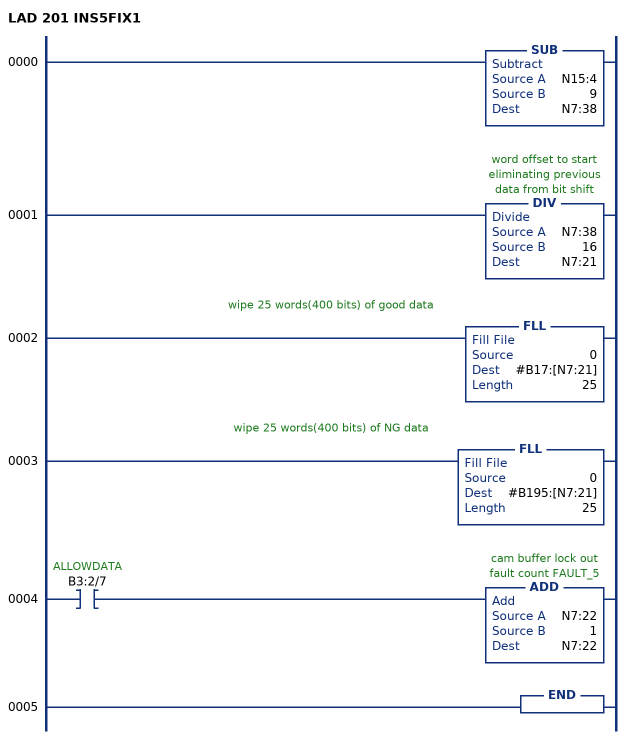
% Rung: 0 %
SOR SUB N15:4 9 N7:38 EOR
%   N15:4  INS_5_TRIG_LOC %
% Rung: 1 %
SOR DIV N7:38 16 N7:21 EOR
%   N7:21  "word offset to start eliminating previous data from bit shift" %
% Rung: 2 %
% wipe 25 words(400 bits) of good data %
SOR FLL 0 #B17:[N7:21] 25 EOR
%   N7:21  "word offset to start eliminating previous data from bit shift" %
% Rung: 3 %
% wipe 25 words(400 bits) of NG data %
SOR FLL 0 #B195:[N7:21] 25 EOR
%   N7:21  "word offset to start eliminating previous data from bit shift" %
% Rung: 4 %
SOR XIC B3:2/7 ADD N7:22 1 N7:22 EOR
%   B3:2/7  ALLOWDATA %
%   N7:22  FAULT_5  "cam buffer lock out fault count" %
% Rung: 5 %
SOR END EOR

LADDER 202 "INS5FIX2"
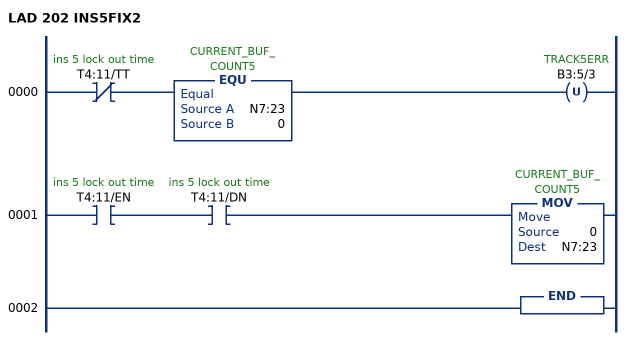
% Rung: 0 %
SOR XIO T4:11/TT EQU N7:23 0 OTU B3:5/3 EOR
%   T4:11  "ins 5 lock out time" %
%   N7:23  CURRENT_BUF_COUNT5 %
%   B3:5/3  TRACK5ERR %
% Rung: 1 %
SOR XIC T4:11/EN XIC T4:11/DN MOV 0 N7:23 EOR
%   T4:11  "ins 5 lock out time" %
%   N7:23  CURRENT_BUF_COUNT5 %
% Rung: 2 %
SOR END EOR

LADDER 203 "HS TRIG5"
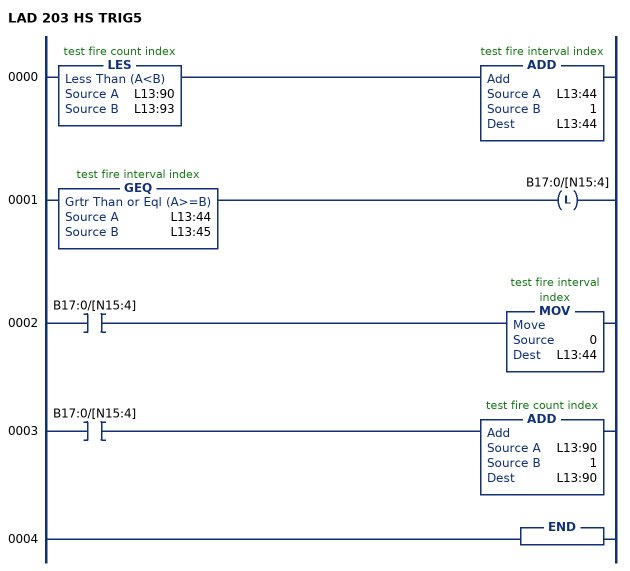
% Rung: 0 %
SOR LES L13:90 L13:93 ADD L13:44 1 L13:44 EOR
%   L13:90  "test fire count index" %
%   L13:93  "test fire count" %
%   L13:44  "test fire interval index" %
% Rung: 1 %
SOR GEQ L13:44 L13:45 OTL B17:0/[N15:4] EOR
%   L13:44  "test fire interval index" %
%   L13:45  "test fire interval" %
%   N15:4  INS_5_TRIG_LOC %
% Rung: 2 %
SOR XIC B17:0/[N15:4] MOV 0 L13:44 EOR
%   N15:4  INS_5_TRIG_LOC %
%   L13:44  "test fire interval index" %
% Rung: 3 %
SOR XIC B17:0/[N15:4] ADD L13:90 1 L13:90 EOR
%   N15:4  INS_5_TRIG_LOC %
%   L13:90  "test fire count index" %
% Rung: 4 %
SOR END EOR

LADDER 212 "INS6"
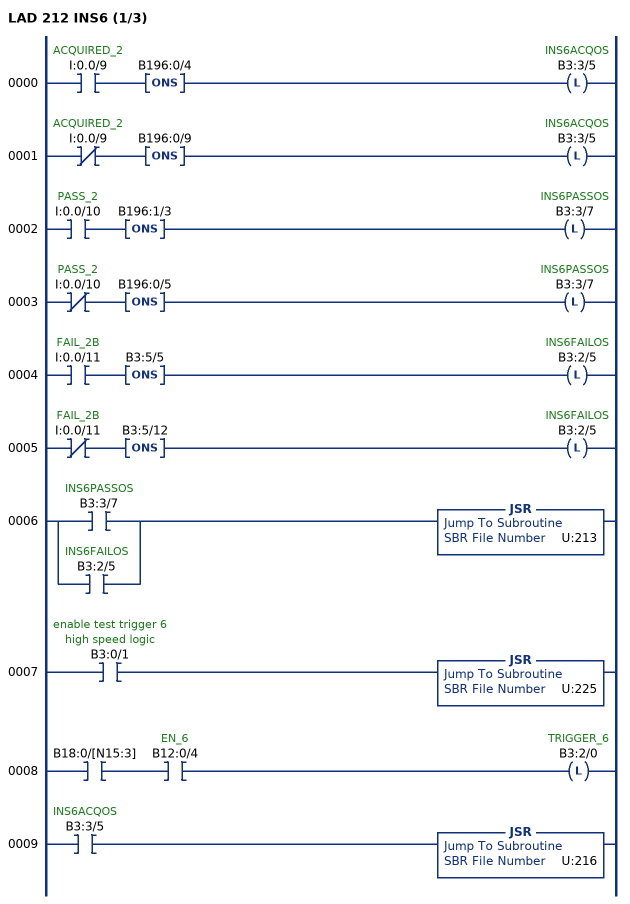
% Rung: 0 %
SOR XIC I:0.0/9 ONS B196:0/4 OTL B3:3/5 EOR
%   I:0.0/9  ACQUIRED_2 %
%   B3:3/5  INS6ACQOS %
% Rung: 1 %
SOR XIO I:0.0/9 ONS B196:0/9 OTL B3:3/5 EOR
%   I:0.0/9  ACQUIRED_2 %
%   B3:3/5  INS6ACQOS %
% Rung: 2 %
SOR XIC I:0.0/10 ONS B196:1/3 OTL B3:3/7 EOR
%   I:0.0/10  PASS_2 %
%   B3:3/7  INS6PASSOS %
% Rung: 3 %
SOR XIO I:0.0/10 ONS B196:0/5 OTL B3:3/7 EOR
%   I:0.0/10  PASS_2 %
%   B3:3/7  INS6PASSOS %
% Rung: 4 %
SOR XIC I:0.0/11 ONS B3:5/5 OTL B3:2/5 EOR
%   I:0.0/11  FAIL_2B %
%   B3:2/5  INS6FAILOS %
% Rung: 5 %
SOR XIO I:0.0/11 ONS B3:5/12 OTL B3:2/5 EOR
%   I:0.0/11  FAIL_2B %
%   B3:2/5  INS6FAILOS %
% Rung: 6 %
SOR BST XIC B3:3/7 NXB XIC B3:2/5 BND JSR U:213 EOR
%   B3:3/7  INS6PASSOS %
%   B3:2/5  INS6FAILOS %
% Rung: 7 %
SOR XIC B3:0/1 JSR U:225 EOR
%   B3:0/1  "enable test trigger 6 high speed logic" %
% Rung: 8 %
SOR XIC B18:0/[N15:3] XIC B12:0/4 OTL B3:2/0 EOR
%   N15:3  INS_6_TRIG_LOC %
%   B12:0/4  EN_6 %
%   B3:2/0  TRIGGER_6 %
% Rung: 9 %
SOR XIC B3:3/5 JSR U:216 EOR
%   B3:3/5  INS6ACQOS %

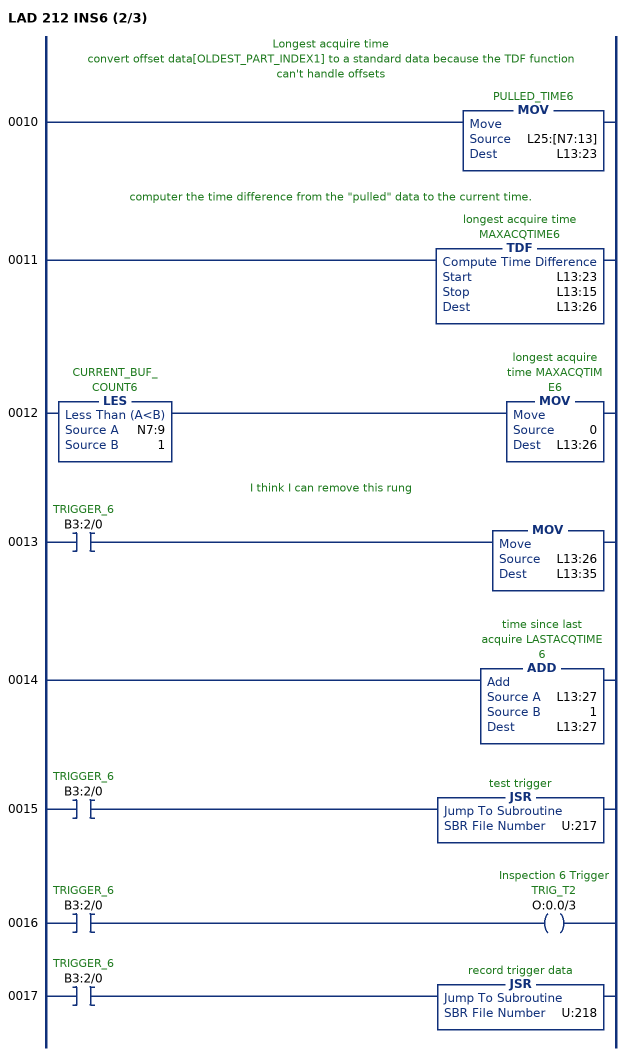
% Rung: 10 %
% Longest acquire time
% convert offset data[OLDEST_PART_INDEX1] to a standard data because the TDF function can't handle offsets %
SOR MOV L25:[N7:13] L13:23 EOR
%   N7:13  OLDEST_PART_INDEX6 %
%   L13:23  PULLED_TIME6 %
% Rung: 11 %
% computer the time difference from the "pulled" data to the current time. %
SOR TDF L13:23 L13:15 L13:26 EOR
%   L13:23  PULLED_TIME6 %
%   L13:15  TOP_TIME %
%   L13:26  MAXACQTIME6  "longest acquire time" %
% Rung: 12 %
SOR LES N7:9 1 MOV 0 L13:26 EOR
%   N7:9  CURRENT_BUF_COUNT6 %
%   L13:26  MAXACQTIME6  "longest acquire time" %
% Rung: 13 %
% I think I can remove this rung %
SOR XIC B3:2/0 MOV L13:26 L13:35 EOR
%   B3:2/0  TRIGGER_6 %
%   L13:26  MAXACQTIME6  "longest acquire time" %
% Rung: 14 %
SOR ADD L13:27 1 L13:27 EOR
%   L13:27  LASTACQTIME6  "time since last acquire" %
% Rung: 15 %
SOR XIC B3:2/0 JSR U:217 EOR
%   B3:2/0  TRIGGER_6 %
%   U:217  "test trigger" %
% Rung: 16 %
SOR XIC B3:2/0 OTE O:0.0/3 EOR
%   B3:2/0  TRIGGER_6 %
%   O:0.0/3  TRIG_T2  "Inspection 6 Trigger" %
% Rung: 17 %
SOR XIC B3:2/0 JSR U:218 EOR
%   B3:2/0  TRIGGER_6 %
%   U:218  "record trigger data" %

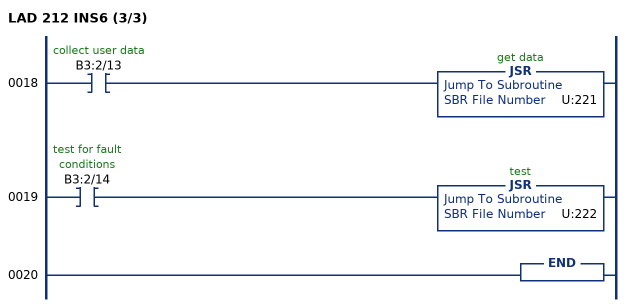
% Rung: 18 %
SOR XIC B3:2/13 JSR U:221 EOR
%   B3:2/13  "collect user data" %
%   U:221  "get data" %
% Rung: 19 %
SOR XIC B3:2/14 JSR U:222 EOR
%   B3:2/14  "test for fault conditions" %
%   U:222  "test" %
% Rung: 20 %
SOR END EOR

LADDER 213 "INS6RESULT"
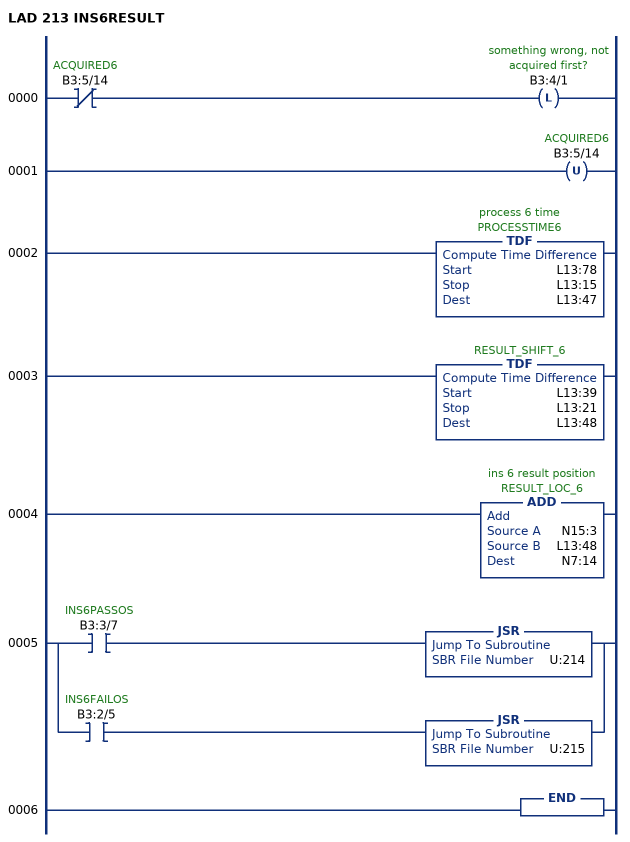
% Rung: 0 %
SOR XIO B3:5/14 OTL B3:4/1 EOR
%   B3:5/14  ACQUIRED6 %
%   B3:4/1  "something wrong, not acquired first?" %
% Rung: 1 %
SOR OTU B3:5/14 EOR
%   B3:5/14  ACQUIRED6 %
% Rung: 2 %
SOR TDF L13:78 L13:15 L13:47 EOR
%   L13:78  TIMEOFACQ6  "the time of the last acquire" %
%   L13:15  TOP_TIME %
%   L13:47  PROCESSTIME6  "process 6 time" %
% Rung: 3 %
SOR TDF L13:39 L13:21 L13:48 EOR
%   L13:39  PROCESS_START_POS_6 %
%   L13:21  TOP_POSITION %
%   L13:48  RESULT_SHIFT_6 %
% Rung: 4 %
SOR ADD N15:3 L13:48 N7:14 EOR
%   N15:3  INS_6_TRIG_LOC %
%   L13:48  RESULT_SHIFT_6 %
%   N7:14  RESULT_LOC_6  "ins 6 result position" %
% Rung: 5 %
SOR BST XIC B3:3/7 JSR U:214 NXB XIC B3:2/5 JSR U:215 BND EOR
%   B3:3/7  INS6PASSOS %
%   B3:2/5  INS6FAILOS %
% Rung: 6 %
SOR END EOR

LADDER 214 "INS6PASS"
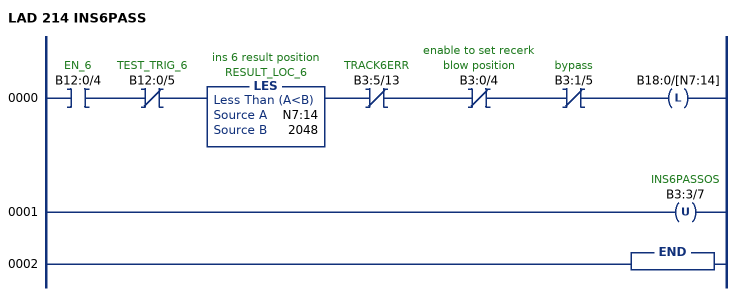
% Rung: 0 %
SOR XIC B12:0/4 XIO B12:0/5 LES N7:14 2048 XIO B3:5/13 XIO B3:0/4 XIO B3:1/5 OTL B18:0/[N7:14] EOR
%   B12:0/4  EN_6 %
%   B12:0/5  TEST_TRIG_6 %
%   N7:14  RESULT_LOC_6  "ins 6 result position" %
%   B3:5/13  TRACK6ERR %
%   B3:0/4  "enable to set recerk blow position" %
%   B3:1/5  "bypass" %
% Rung: 1 %
SOR OTU B3:3/7 EOR
%   B3:3/7  INS6PASSOS %
% Rung: 2 %
SOR END EOR

LADDER 215 "INS6FAIL"
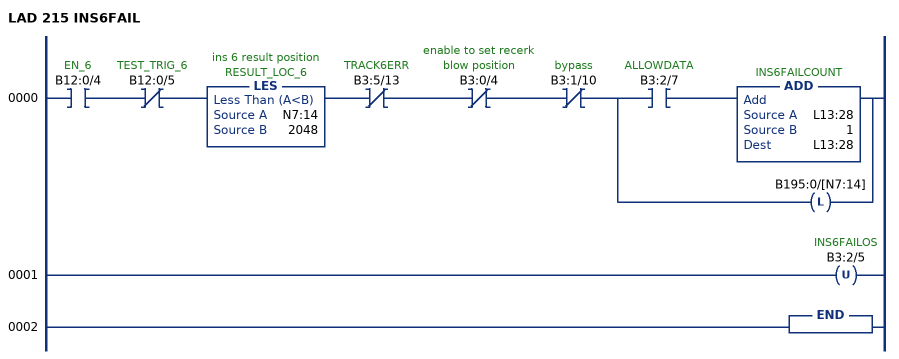
% Rung: 0 %
SOR XIC B12:0/4 XIO B12:0/5 LES N7:14 2048 XIO B3:5/13 XIO B3:0/4 XIO B3:1/10 BST XIC B3:2/7 ADD L13:28 1 L13:28 NXB OTL B195:0/[N7:14] BND EOR
%   B12:0/4  EN_6 %
%   B12:0/5  TEST_TRIG_6 %
%   N7:14  RESULT_LOC_6  "ins 6 result position" %
%   B3:5/13  TRACK6ERR %
%   B3:0/4  "enable to set recerk blow position" %
%   B3:1/10  "bypass" %
%   B3:2/7  ALLOWDATA %
%   L13:28  INS6FAILCOUNT %
% Rung: 1 %
SOR OTU B3:2/5 EOR
%   B3:2/5  INS6FAILOS %
% Rung: 2 %
SOR END EOR

LADDER 216 "INS6ACQ"
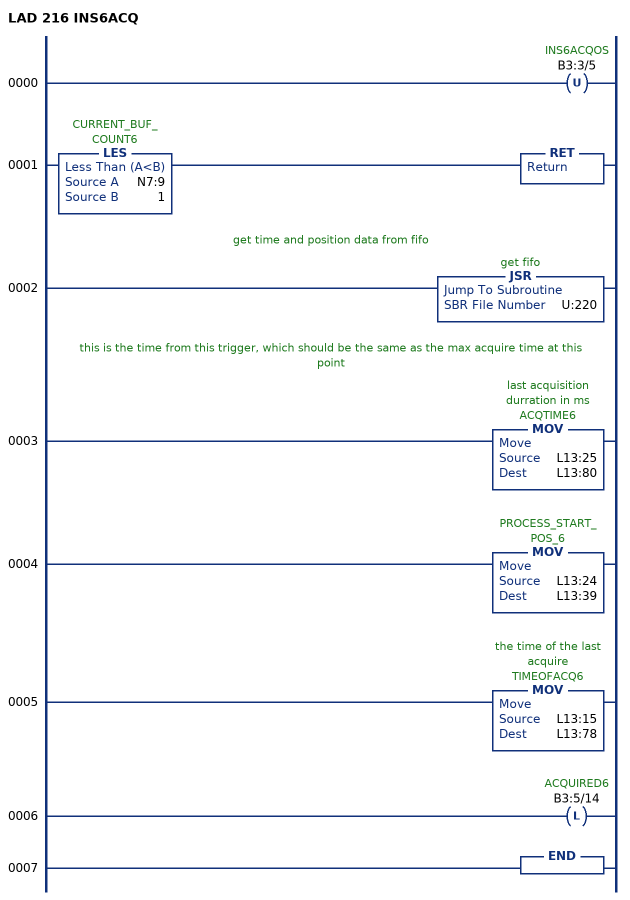
% Rung: 0 %
SOR OTU B3:3/5 EOR
%   B3:3/5  INS6ACQOS %
% Rung: 1 %
SOR LES N7:9 1 RET EOR
%   N7:9  CURRENT_BUF_COUNT6 %
% Rung: 2 %
% get time and position data from fifo %
SOR JSR U:220 EOR
%   U:220  "get fifo" %
% Rung: 3 %
% this is the time from this trigger, which should be the same as the max acquire time at this point %
SOR MOV L13:25 L13:80 EOR
%   L13:25  TIME_SPAN6 %
%   L13:80  ACQTIME6  "last acquisition durration in ms" %
% Rung: 4 %
SOR MOV L13:24 L13:39 EOR
%   L13:24  PULLED_POSITION6 %
%   L13:39  PROCESS_START_POS_6 %
% Rung: 5 %
SOR MOV L13:15 L13:78 EOR
%   L13:15  TOP_TIME %
%   L13:78  TIMEOFACQ6  "the time of the last acquire" %
% Rung: 6 %
SOR OTL B3:5/14 EOR
%   B3:5/14  ACQUIRED6 %
% Rung: 7 %
SOR END EOR

LADDER 217 "Q6TIMETEST"
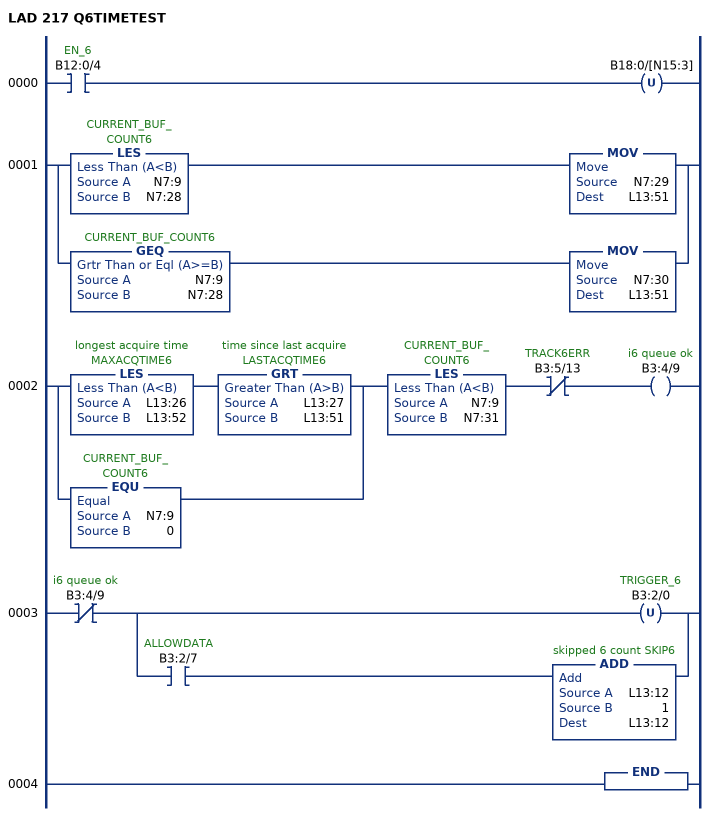
% Rung: 0 %
SOR XIC B12:0/4 OTU B18:0/[N15:3] EOR
%   B12:0/4  EN_6 %
%   N15:3  INS_6_TRIG_LOC %
% Rung: 1 %
SOR BST LES N7:9 N7:28 MOV N7:29 L13:51 NXB GEQ N7:9 N7:28 MOV N7:30 L13:51 BND EOR
%   N7:9  CURRENT_BUF_COUNT6 %
% Rung: 2 %
SOR BST LES L13:26 L13:52 GRT L13:27 L13:51 NXB EQU N7:9 0 BND LES N7:9 N7:31 XIO B3:5/13 OTE B3:4/9 EOR
%   L13:26  MAXACQTIME6  "longest acquire time" %
%   L13:52  ACQTIMELIMIT6 %
%   L13:27  LASTACQTIME6  "time since last acquire" %
%   N7:9  CURRENT_BUF_COUNT6 %
%   N7:31  "maximum buffers" %
%   B3:5/13  TRACK6ERR %
%   B3:4/9  "i6 queue ok" %
% Rung: 3 %
SOR XIO B3:4/9 BST OTU B3:2/0 NXB XIC B3:2/7 ADD L13:12 1 L13:12 BND EOR
%   B3:4/9  "i6 queue ok" %
%   B3:2/0  TRIGGER_6 %
%   B3:2/7  ALLOWDATA %
%   L13:12  SKIP6  "skipped 6 count" %
% Rung: 4 %
SOR END EOR

LADDER 218 "INS6TRIG"
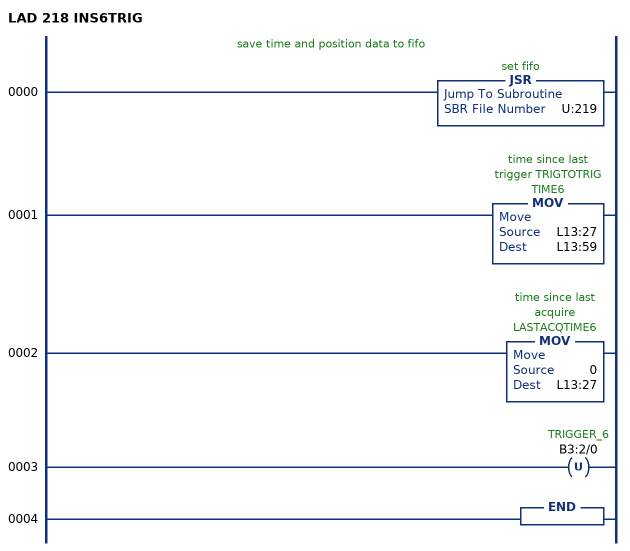
% Rung: 0 %
% save time and position data to fifo %
SOR JSR U:219 EOR
%   U:219  "set fifo" %
% Rung: 1 %
SOR MOV L13:27 L13:59 EOR
%   L13:27  LASTACQTIME6  "time since last acquire" %
%   L13:59  TRIGTOTRIGTIME6  "time since last trigger" %
% Rung: 2 %
SOR MOV 0 L13:27 EOR
%   L13:27  LASTACQTIME6  "time since last acquire" %
% Rung: 3 %
SOR OTU B3:2/0 EOR
%   B3:2/0  TRIGGER_6 %
% Rung: 4 %
SOR END EOR

LADDER 219 "FIFO6SET"
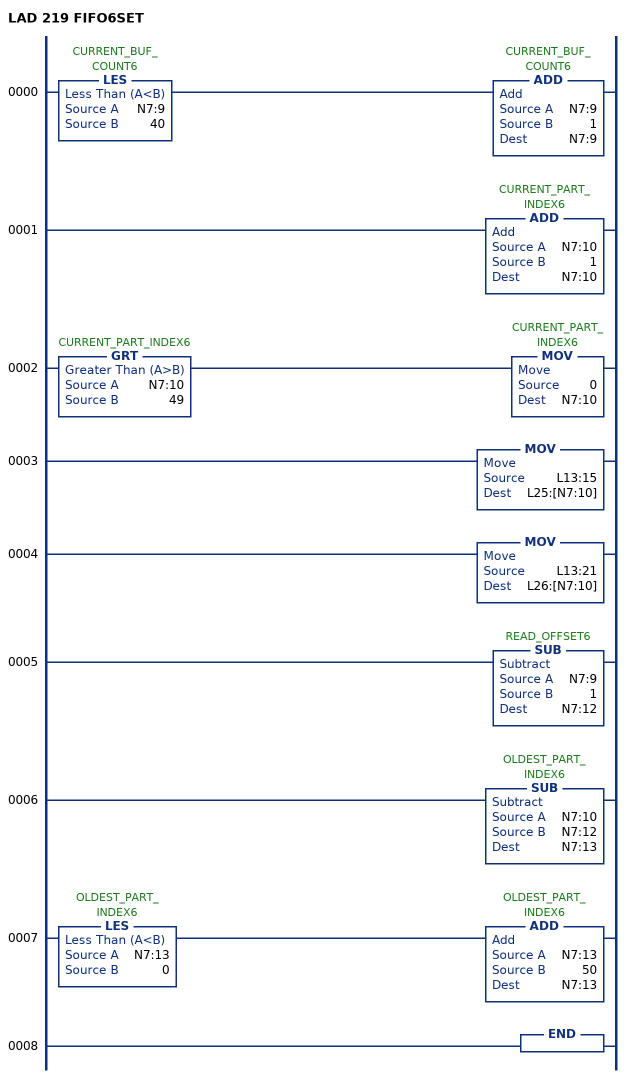
% Rung: 0 %
SOR LES N7:9 40 ADD N7:9 1 N7:9 EOR
%   N7:9  CURRENT_BUF_COUNT6 %
% Rung: 1 %
SOR ADD N7:10 1 N7:10 EOR
%   N7:10  CURRENT_PART_INDEX6 %
% Rung: 2 %
SOR GRT N7:10 49 MOV 0 N7:10 EOR
%   N7:10  CURRENT_PART_INDEX6 %
% Rung: 3 %
SOR MOV L13:15 L25:[N7:10] EOR
%   L13:15  TOP_TIME %
%   N7:10  CURRENT_PART_INDEX6 %
% Rung: 4 %
SOR MOV L13:21 L26:[N7:10] EOR
%   L13:21  TOP_POSITION %
%   N7:10  CURRENT_PART_INDEX6 %
% Rung: 5 %
SOR SUB N7:9 1 N7:12 EOR
%   N7:9  CURRENT_BUF_COUNT6 %
%   N7:12  "READ_OFFSET6" %
% Rung: 6 %
SOR SUB N7:10 N7:12 N7:13 EOR
%   N7:10  CURRENT_PART_INDEX6 %
%   N7:12  "READ_OFFSET6" %
%   N7:13  OLDEST_PART_INDEX6 %
% Rung: 7 %
SOR LES N7:13 0 ADD N7:13 50 N7:13 EOR
%   N7:13  OLDEST_PART_INDEX6 %
% Rung: 8 %
SOR END EOR

LADDER 220 "FIFO6GET"
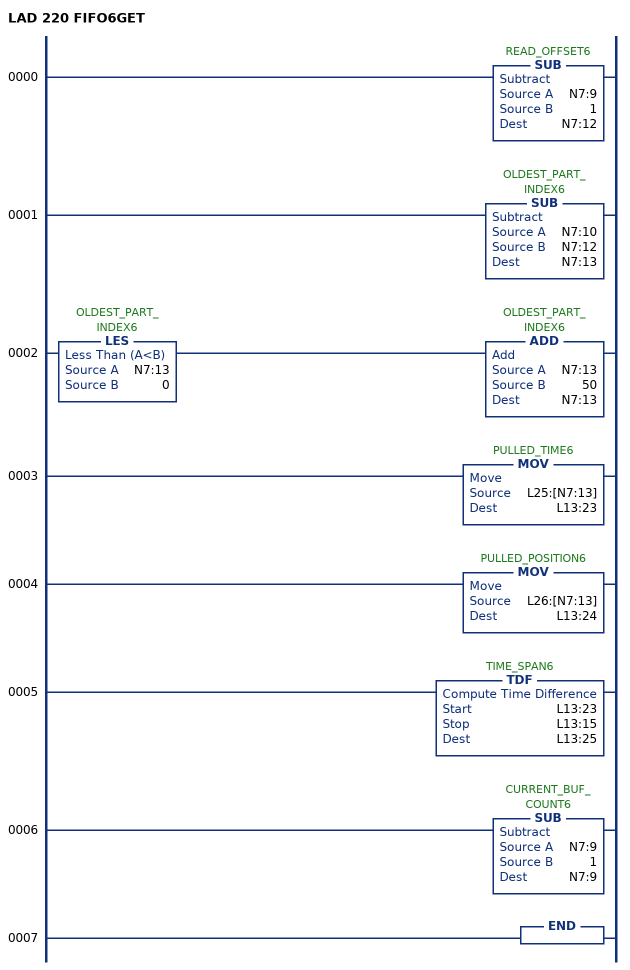
% Rung: 0 %
SOR SUB N7:9 1 N7:12 EOR
%   N7:9  CURRENT_BUF_COUNT6 %
%   N7:12  "READ_OFFSET6" %
% Rung: 1 %
SOR SUB N7:10 N7:12 N7:13 EOR
%   N7:10  CURRENT_PART_INDEX6 %
%   N7:12  "READ_OFFSET6" %
%   N7:13  OLDEST_PART_INDEX6 %
% Rung: 2 %
SOR LES N7:13 0 ADD N7:13 50 N7:13 EOR
%   N7:13  OLDEST_PART_INDEX6 %
% Rung: 3 %
SOR MOV L25:[N7:13] L13:23 EOR
%   N7:13  OLDEST_PART_INDEX6 %
%   L13:23  PULLED_TIME6 %
% Rung: 4 %
SOR MOV L26:[N7:13] L13:24 EOR
%   N7:13  OLDEST_PART_INDEX6 %
%   L13:24  PULLED_POSITION6 %
% Rung: 5 %
SOR TDF L13:23 L13:15 L13:25 EOR
%   L13:23  PULLED_TIME6 %
%   L13:15  TOP_TIME %
%   L13:25  TIME_SPAN6 %
% Rung: 6 %
SOR SUB N7:9 1 N7:9 EOR
%   N7:9  CURRENT_BUF_COUNT6 %
% Rung: 7 %
SOR END EOR

LADDER 221 "INSDATA6"
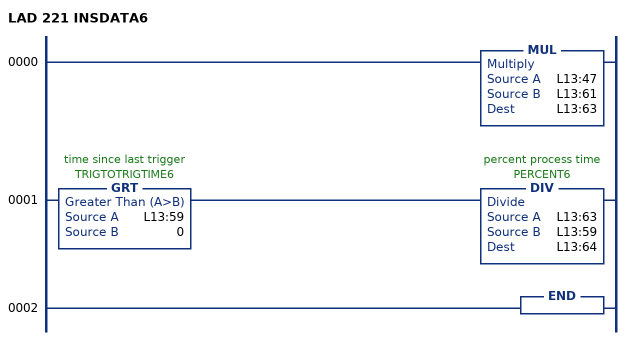
% Rung: 0 %
SOR MUL L13:47 L13:61 L13:63 EOR
%   L13:47  PROCESSTIME6  "process 6 time" %
%   L13:61  "max acquisition time in ms" %
% Rung: 1 %
SOR GRT L13:59 0 DIV L13:63 L13:59 L13:64 EOR
%   L13:59  TRIGTOTRIGTIME6  "time since last trigger" %
%   L13:64  PERCENT6  "percent process time" %
% Rung: 2 %
SOR END EOR

LADDER 222 "TESTFAULT6"
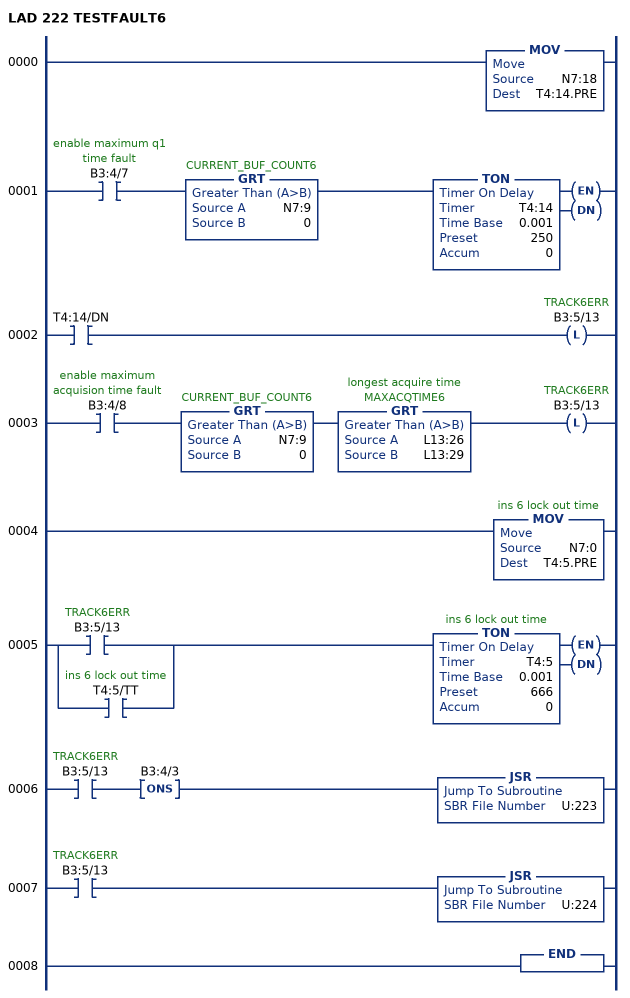
% Rung: 0 %
SOR MOV N7:18 T4:14.PRE EOR
%   N7:18  "max allowed ms time for q to be above 1 if safe fault is used" %
% Rung: 1 %
SOR XIC B3:4/7 GRT N7:9 0 TON T4:14 0.001 250 0 EOR
%   B3:4/7  "enable maximum q1 time fault" %
%   N7:9  CURRENT_BUF_COUNT6 %
% Rung: 2 %
SOR XIC T4:14/DN OTL B3:5/13 EOR
%   B3:5/13  TRACK6ERR %
% Rung: 3 %
SOR XIC B3:4/8 GRT N7:9 0 GRT L13:26 L13:29 OTL B3:5/13 EOR
%   B3:4/8  "enable maximum acquision time fault" %
%   N7:9  CURRENT_BUF_COUNT6 %
%   L13:26  MAXACQTIME6  "longest acquire time" %
%   L13:29  "maximum of the longest acquire time allowed if maximum acquire time fault is enabled" %
%   B3:5/13  TRACK6ERR %
% Rung: 4 %
SOR MOV N7:0 T4:5.PRE EOR
%   N7:0  "ms time setting to lock out inspection to give all pending images a chance to clear" %
%   T4:5  "ins 6 lock out time" %
% Rung: 5 %
SOR BST XIC B3:5/13 NXB XIC T4:5/TT BND TON T4:5 0.001 666 0 EOR
%   B3:5/13  TRACK6ERR %
%   T4:5  "ins 6 lock out time" %
% Rung: 6 %
SOR XIC B3:5/13 ONS B3:4/3 JSR U:223 EOR
%   B3:5/13  TRACK6ERR %
% Rung: 7 %
SOR XIC B3:5/13 JSR U:224 EOR
%   B3:5/13  TRACK6ERR %
% Rung: 8 %
SOR END EOR

LADDER 223 "INS6FIX1"
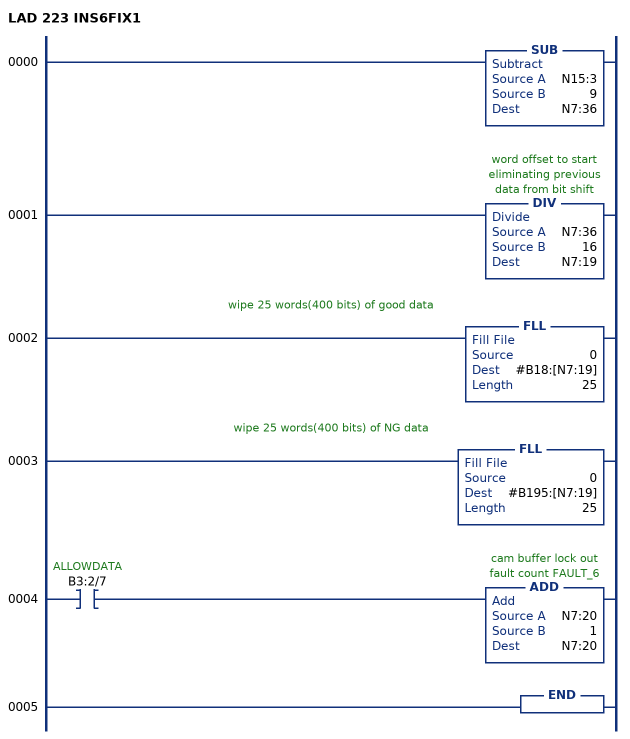
% Rung: 0 %
SOR SUB N15:3 9 N7:36 EOR
%   N15:3  INS_6_TRIG_LOC %
% Rung: 1 %
SOR DIV N7:36 16 N7:19 EOR
%   N7:19  "word offset to start eliminating previous data from bit shift" %
% Rung: 2 %
% wipe 25 words(400 bits) of good data %
SOR FLL 0 #B18:[N7:19] 25 EOR
%   N7:19  "word offset to start eliminating previous data from bit shift" %
% Rung: 3 %
% wipe 25 words(400 bits) of NG data %
SOR FLL 0 #B195:[N7:19] 25 EOR
%   N7:19  "word offset to start eliminating previous data from bit shift" %
% Rung: 4 %
SOR XIC B3:2/7 ADD N7:20 1 N7:20 EOR
%   B3:2/7  ALLOWDATA %
%   N7:20  FAULT_6  "cam buffer lock out fault count" %
% Rung: 5 %
SOR END EOR

LADDER 224 "INS6FIX2"
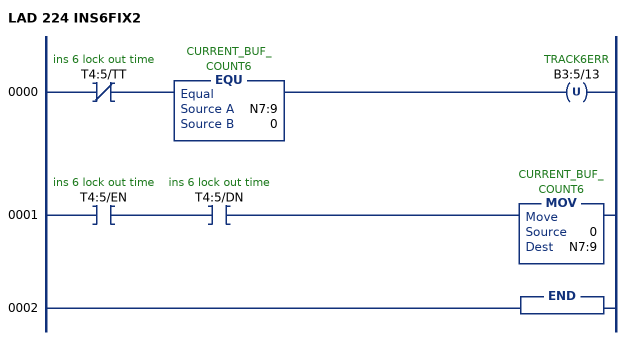
% Rung: 0 %
SOR XIO T4:5/TT EQU N7:9 0 OTU B3:5/13 EOR
%   T4:5  "ins 6 lock out time" %
%   N7:9  CURRENT_BUF_COUNT6 %
%   B3:5/13  TRACK6ERR %
% Rung: 1 %
SOR XIC T4:5/EN XIC T4:5/DN MOV 0 N7:9 EOR
%   T4:5  "ins 6 lock out time" %
%   N7:9  CURRENT_BUF_COUNT6 %
% Rung: 2 %
SOR END EOR

LADDER 225 "HS TRIG6"
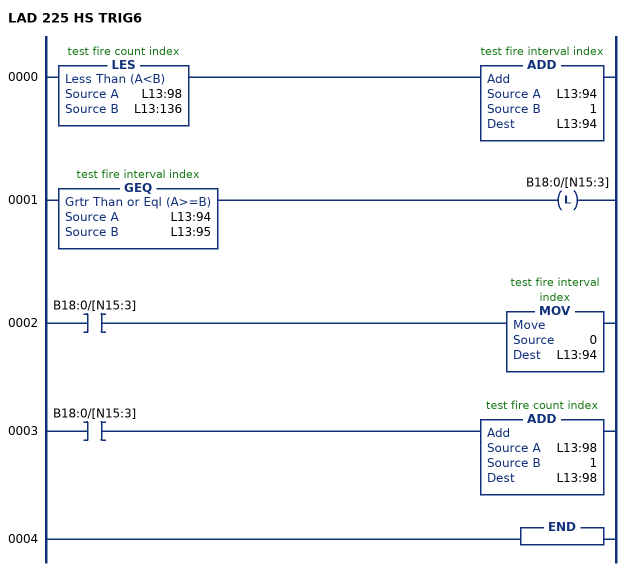
% Rung: 0 %
SOR LES L13:98 L13:136 ADD L13:94 1 L13:94 EOR
%   L13:98  "test fire count index" %
%   L13:136  "test fire count" %
%   L13:94  "test fire interval index" %
% Rung: 1 %
SOR GEQ L13:94 L13:95 OTL B18:0/[N15:3] EOR
%   L13:94  "test fire interval index" %
%   L13:95  "test fire interval" %
%   N15:3  INS_6_TRIG_LOC %
% Rung: 2 %
SOR XIC B18:0/[N15:3] MOV 0 L13:94 EOR
%   N15:3  INS_6_TRIG_LOC %
%   L13:94  "test fire interval index" %
% Rung: 3 %
SOR XIC B18:0/[N15:3] ADD L13:98 1 L13:98 EOR
%   N15:3  INS_6_TRIG_LOC %
%   L13:98  "test fire count index" %
% Rung: 4 %
SOR END EOR

LADDER 240 "PASS BLOW"
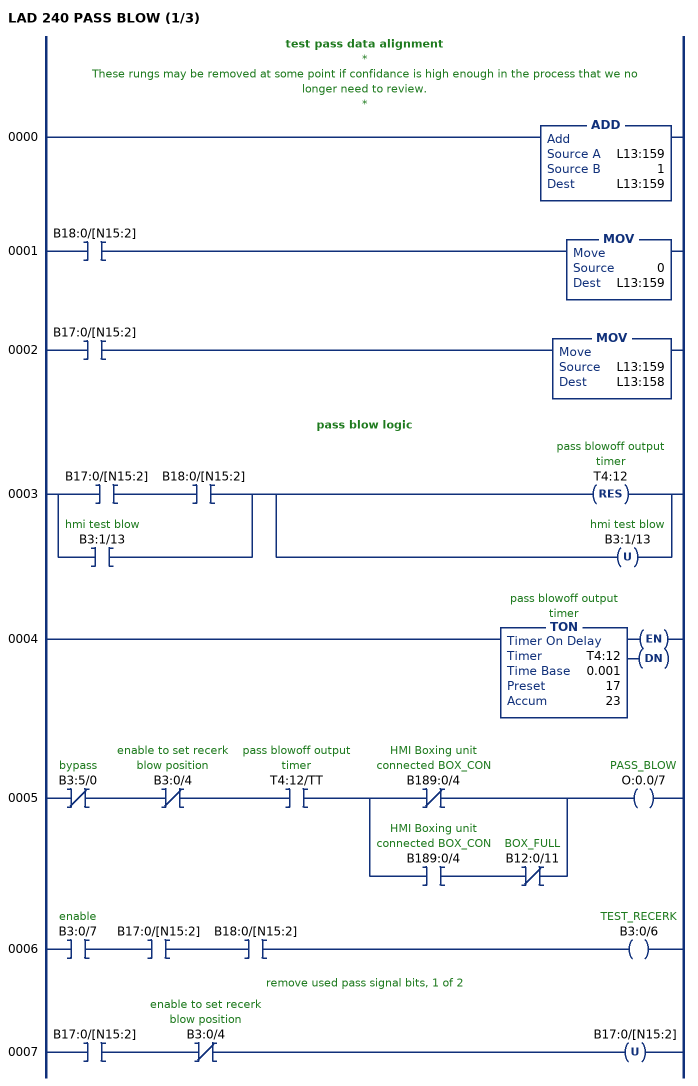
% Rung: 0 %
% TITLE: test pass data alignment %
% *
% These rungs may be removed at some point if confidance is high enough in the process that we no longer need to review.
% * %
SOR ADD L13:159 1 L13:159 EOR
% Rung: 1 %
SOR XIC B18:0/[N15:2] MOV 0 L13:159 EOR
%   N15:2  BLOW_PT %
% Rung: 2 %
SOR XIC B17:0/[N15:2] MOV L13:159 L13:158 EOR
%   N15:2  BLOW_PT %
% Rung: 3 %
% TITLE: pass blow logic %
SOR BST XIC B17:0/[N15:2] XIC B18:0/[N15:2] NXB XIC B3:1/13 BND BST RES T4:12 NXB OTU B3:1/13 BND EOR
%   N15:2  BLOW_PT %
%   B3:1/13  "hmi test blow" %
%   T4:12  "pass blowoff output timer" %
% Rung: 4 %
SOR TON T4:12 0.001 17 23 EOR
%   T4:12  "pass blowoff output timer" %
% Rung: 5 %
SOR XIO B3:5/0 XIO B3:0/4 XIC T4:12/TT BST XIO B189:0/4 NXB XIC B189:0/4 XIO B12:0/11 BND OTE O:0.0/7 EOR
%   B3:5/0  "bypass" %
%   B3:0/4  "enable to set recerk blow position" %
%   T4:12  "pass blowoff output timer" %
%   B189:0/4  BOX_CON  "HMI Boxing unit connected" %
%   B12:0/11  BOX_FULL %
%   O:0.0/7  PASS_BLOW %
% Rung: 6 %
SOR XIC B3:0/7 XIC B17:0/[N15:2] XIC B18:0/[N15:2] OTE B3:0/6 EOR
%   B3:0/7  "enable" %
%   N15:2  BLOW_PT %
%   B3:0/6  TEST_RECERK %
% Rung: 7 %
% remove used pass signal bits, 1 of 2 %
SOR XIC B17:0/[N15:2] XIO B3:0/4 OTU B17:0/[N15:2] EOR
%   N15:2  BLOW_PT %
%   B3:0/4  "enable to set recerk blow position" %

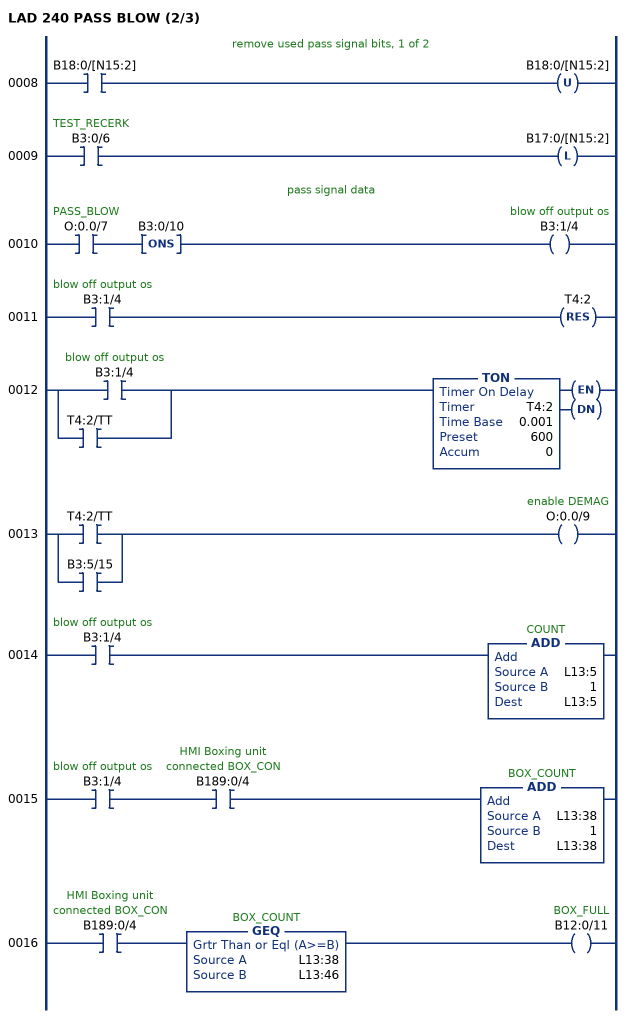
% Rung: 8 %
% remove used pass signal bits, 1 of 2 %
SOR XIC B18:0/[N15:2] OTU B18:0/[N15:2] EOR
%   N15:2  BLOW_PT %
% Rung: 9 %
SOR XIC B3:0/6 OTL B17:0/[N15:2] EOR
%   B3:0/6  TEST_RECERK %
%   N15:2  BLOW_PT %
% Rung: 10 %
% pass signal data %
SOR XIC O:0.0/7 ONS B3:0/10 OTE B3:1/4 EOR
%   O:0.0/7  PASS_BLOW %
%   B3:1/4  "blow off output os" %
% Rung: 11 %
SOR XIC B3:1/4 RES T4:2 EOR
%   B3:1/4  "blow off output os" %
% Rung: 12 %
SOR BST XIC B3:1/4 NXB XIC T4:2/TT BND TON T4:2 0.001 600 0 EOR
%   B3:1/4  "blow off output os" %
% Rung: 13 %
SOR BST XIC T4:2/TT NXB XIC B3:5/15 BND OTE O:0.0/9 EOR
%   O:0.0/9  DEMAG  "enable" %
% Rung: 14 %
SOR XIC B3:1/4 ADD L13:5 1 L13:5 EOR
%   B3:1/4  "blow off output os" %
%   L13:5  COUNT %
% Rung: 15 %
SOR XIC B3:1/4 XIC B189:0/4 ADD L13:38 1 L13:38 EOR
%   B3:1/4  "blow off output os" %
%   B189:0/4  BOX_CON  "HMI Boxing unit connected" %
%   L13:38  BOX_COUNT %
% Rung: 16 %
SOR XIC B189:0/4 GEQ L13:38 L13:46 OTE B12:0/11 EOR
%   B189:0/4  BOX_CON  "HMI Boxing unit connected" %
%   L13:38  BOX_COUNT %
%   L13:46  BOX_LIMIT  "box count setpoint" %
%   B12:0/11  BOX_FULL %

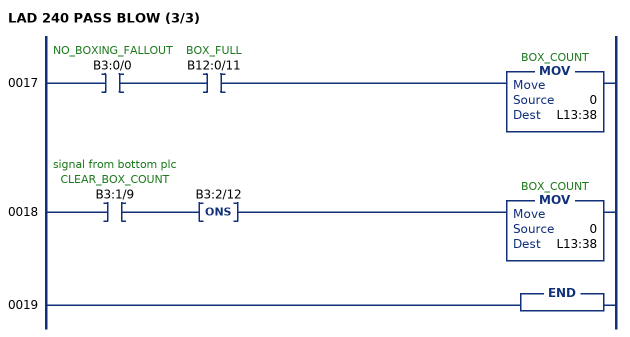
% Rung: 17 %
SOR XIC B3:0/0 XIC B12:0/11 MOV 0 L13:38 EOR
%   B3:0/0  NO_BOXING_FALLOUT %
%   B12:0/11  BOX_FULL %
%   L13:38  BOX_COUNT %
% Rung: 18 %
SOR XIC B3:1/9 ONS B3:2/12 MOV 0 L13:38 EOR
%   B3:1/9  CLEAR_BOX_COUNT  "signal from bottom plc" %
%   L13:38  BOX_COUNT %
% Rung: 19 %
SOR END EOR

LADDER 242 "RECERK"
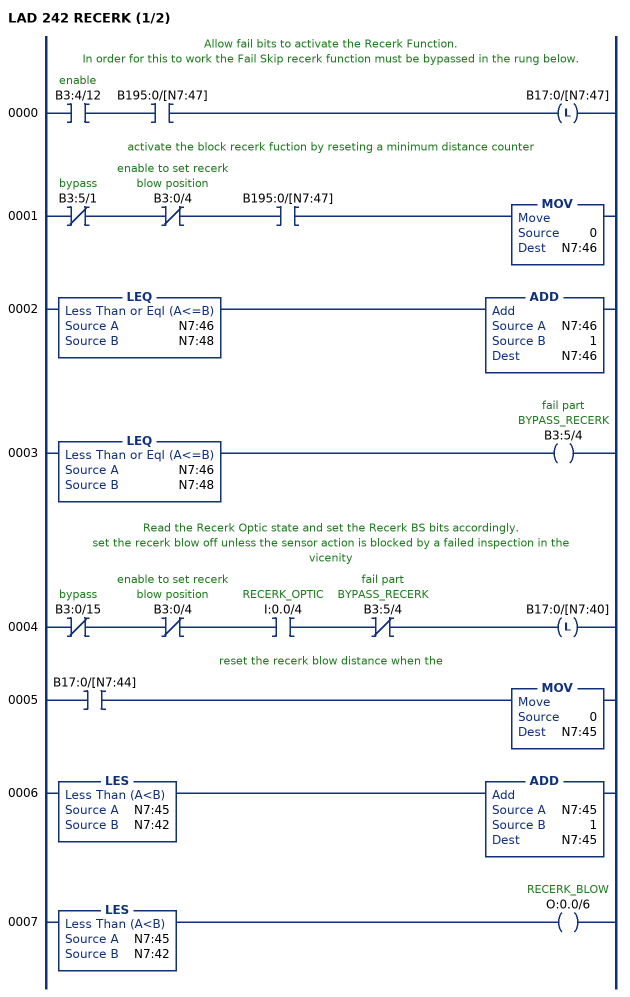
% Rung: 0 %
% Allow fail bits to activate the Recerk Function.
% In order for this to work the Fail Skip recerk function must be bypassed in the rung below. %
SOR XIC B3:4/12 XIC B195:0/[N7:47] OTL B17:0/[N7:47] EOR
%   B3:4/12  "enable" %
%   N7:47  RECERK_BLOCKOPTIC_PT %
% Rung: 1 %
% activate the block recerk fuction by reseting a minimum distance counter %
SOR XIO B3:5/1 XIO B3:0/4 XIC B195:0/[N7:47] MOV 0 N7:46 EOR
%   B3:5/1  "bypass" %
%   B3:0/4  "enable to set recerk blow position" %
%   N7:47  RECERK_BLOCKOPTIC_PT %
% Rung: 2 %
SOR LEQ N7:46 N7:48 ADD N7:46 1 N7:46 EOR
%   N7:48  RECERK_BLK_BLOW_DIST %
% Rung: 3 %
SOR LEQ N7:46 N7:48 OTE B3:5/4 EOR
%   N7:48  RECERK_BLK_BLOW_DIST %
%   B3:5/4  BYPASS_RECERK  "fail part" %
% Rung: 4 %
% Read the Recerk Optic state and set the Recerk BS bits accordingly.
% 
% set the recerk blow off unless the sensor action is blocked by a failed inspection in the vicenity %
SOR XIO B3:0/15 XIO B3:0/4 XIC I:0.0/4 XIO B3:5/4 OTL B17:0/[N7:40] EOR
%   B3:0/15  "bypass" %
%   B3:0/4  "enable to set recerk blow position" %
%   I:0.0/4  RECERK_OPTIC %
%   B3:5/4  BYPASS_RECERK  "fail part" %
%   N7:40  RECERK_OPTIC_POS %
% Rung: 5 %
% reset the recerk blow distance when the %
SOR XIC B17:0/[N7:44] MOV 0 N7:45 EOR
%   N7:44  RECERK_BLOW_POS  "adjusted for blow length" %
% Rung: 6 %
SOR LES N7:45 N7:42 ADD N7:45 1 N7:45 EOR
%   N7:42  RECERK_BLOW_LENGTH %
% Rung: 7 %
SOR LES N7:45 N7:42 OTE O:0.0/6 EOR
%   N7:42  RECERK_BLOW_LENGTH %
%   O:0.0/6  RECERK_BLOW %

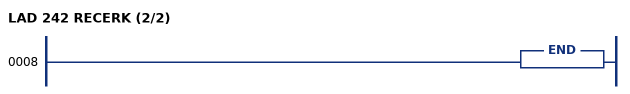
% Rung: 8 %
SOR END EOR

LADDER 243 "RECERK SET"
